(*
SPDX-FileCopyrightText: © 2026 Oleksandr Tiutyk <trofimich@gmail.com>
SPDX-License-Identifier: MIT
License: https://opensource.org/license/mit
*)

FUNCTION_BLOCK DemoExceptionGenerator EXTENDS TOF_Automation.InputLeafAutomationComponent IMPLEMENTS IDemoExceptionGenerator
VAR_STAT
	//! <summary>Class name shared by all instances of this function block.</summary>
	{attribute 'hide'} 
	_ClassName : STRING := __POUNAME();
END_VAR
VAR
	_ExceptionMessage : STRING(255);
	_IsCritical : BOOL;
 	
	_Throw : BOOL; 	
END_VAR

{attribute 'monitoring' := 'call'}
PROPERTY ClassName : REFERENCE TO STRING
GET
ClassName REF= _ClassName;
END_GET
END_PROPERTY

{attribute 'monitoring' := 'call'}
PROPERTY NamespaceName : REFERENCE TO STRING
GET
NamespaceName REF= CurrentNamespace.Name;
END_GET
END_PROPERTY

METHOD PROTECTED OnProcessInput
VAR
	exceptionMessage : STRING(255);
END_VAR
VAR
	demoException : DemoException;
END_VAR
IF _Throw THEN
	_Throw := FALSE;

	exceptionMessage := SEL(_ExceptionMessage = '', _ExceptionMessage, '<empty message>');
		
	demoException.Throw(
		sourceNamespaceName := NamespaceName,
		sourceClassName := ClassName,
		sourcePOUName := __POUNAME(),
		sourcePosition := __POSITION(),
		isCritical := _IsCritical,
		message := exceptionMessage
	);
END_IF
END_METHOD

{attribute 'monitoring' := 'call'}
PROPERTY SelfSize : ULINT
GET
SelfSize := XSIZEOF(THIS^);
END_GET
END_PROPERTY

METHOD ThrowException
VAR_IN_OUT CONSTANT
	exceptionMessage : STRING(255);
	isCritical : BOOL; 
END_VAR
_ExceptionMessage := exceptionMessage;
_IsCritical := isCritical; 	
_Throw := TRUE;
END_METHOD

END_FUNCTION_BLOCK

(* stored: Version 1.1.0.1
   POU DemoExceptionGenerator: Id {45653e5b-ddb2-4268-a8bb-8203bd23d851}, SpecialFunc None
   Folder Commands: Id {9a243b6c-bb40-4290-ad35-0d041c27feab}
   Folder Overriden methods: Id {3ef428ad-b326-4255-bf0a-55ecde7d95c5}
   Property ClassName: Id {0c49b231-cfa2-4c30-95fb-dcb49a96a631}
   Get Get: Id {364b699c-1a13-4a6f-b218-efb219d26924}
   Property NamespaceName: Id {8b36a711-a8d3-4bd9-af14-2fc9e45960ed}
   Get Get: Id {e3321c82-0746-4f2a-a5e9-5339a7f3aeae}
   Method OnProcessInput: Id {467f071b-368d-4346-8295-08235916d67a}
   Property SelfSize: Id {b23aa0bf-c2e5-4bd6-9603-0b1e935641dc}
   Get Get: Id {ec337281-8132-429d-b620-5664fc856c50}
   Method ThrowException: Id {6bb9feb2-1a47-43e2-b743-016cc356f536} *)
